TYPE "MEStoPLC_Common_ext"
VERSION : 0.1
   STRUCT
      "M-HeartBeat" : Bool;
   END_STRUCT;

END_TYPE

